// TwinCAT 3 PLC project PLC_SLAVE
// ProgramVersion: 3.1.4026.16
// libraries:
//   Tc2_Standard, * (Beckhoff Automation GmbH)
//   Tc2_System, * (Beckhoff Automation GmbH)
// project tree:
//   / PlcTask.TcTTO
//   POUs/ MAIN.TcPOU
// real-time tasks:
//   TASK PlcTask: cycle T#1ms, priority 20, ADS port 350
// I/O:
//   DEVICE Device 4 (EtherCAT Slave), AmsNetId 10.200.70.1.5.255
// variable links:
//   PLC_SLAVE Instance <-> Device 4 (EtherCAT Slave)
//     PlcTask Inputs/MAIN.bTrigger <-> Inputs/bTrigger
//     PlcTask Inputs/MAIN.iMasterCounter <-> Inputs/iMasterCounter
//     PlcTask Inputs/MAIN.lrMasterTemp <-> Inputs/lrMasterTemp
//     PlcTask Outputs/MAIN.bFlag <-> Outputs/bFlag
//     PlcTask Outputs/MAIN.iSlaveCounter <-> Outputs/iSlaveCounter
//     PlcTask Outputs/MAIN.lrSlaveTemp <-> Outputs/lrSlaveTemp

CONFIGURATION PLC_SLAVE
    RESOURCE PLC ON TwinCAT3
        TASK PlcTask(INTERVAL := T#2ms, PRIORITY := 20);
        PROGRAM MAIN WITH PlcTask : MAIN;
    END_RESOURCE
END_CONFIGURATION

// ---- POUs/MAIN.TcPOU
PROGRAM MAIN //EtherCAT Slave side
VAR
iMasterCounter 	AT %I* : INT;	//integer 	input from Master
lrMasterTemp 	AT %I* : LREAL;	//lreal		input from Master
bTrigger 		AT %I* : BOOL;	//bool 		input from Master

iSlaveCounter 	AT %Q* : INT;	//integer	output to Master
lrSlaveTemp 	AT %Q* : LREAL;	//lreal		output to Master
bFlag 			AT %Q* : BOOL;	//bool		output to Master

timer1 : TON;
END_VAR

//EtherCAT Slave side
iSlaveCounter 	:= iMasterCounter;
lrSlaveTemp 	:= lrMasterTemp * 2.0;
timer1(	IN:= bTrigger, 
		PT:= T#2S, 
		Q=> bFlag, ET=> );

END_PROGRAM
